{attribute 'qualified_only'}
{attribute 'strict'}
TYPE Color : 
(
	White := 0,
	Black,
	Red,
	Green,
	Blue
) ;
END_TYPE

(* stored: DUT Color: Id f418b0e5-2a53-4d43-a953-dbd4a0200b91 *)
